// TIA Portal V17 export
// export: Created 2025-08-05T09:36:00.9032134Z, ExportSetting WithDefaults, DisplayName Totally Integrated Automation Portal, DisplayVersion V17, DisplayName TIA Portal Openness, DisplayVersion V17, DisplayName TIA Portal Version Control Interface, DisplayVersion V17, DisplayName SINAMICS Startdrive Advanced, DisplayVersion V17, DisplayName SINAMICS Startdrive G130, G150, S120, S150, SINAMICS MV, S210, DisplayVersion V17, DisplayName SINAMICS Startdrive G110M, G120, G120C, G120D, G120P, G115D, DisplayVersion V17, DisplayName STEP 7 Professional, DisplayVersion V17, DisplayName STEP 7 Safety, DisplayVersion V17, DisplayName WinCC Advanced, DisplayVersion V17
TYPE "typeTeststoppSBTPopUpWarn"
// V 01.00
// stored: IsFailsafeCompliant false
   STRUCT
      DoNotOpenSafeGuard : Bool;   // Bremsentest/Teststopp aktiv => Schutzeinrichtung nicht unterbrechen/öffnen / Brake test/test stop active => do not interrupt/open safeguard
      SafeGuardNotOpen { S7_SetPoint := 'True'} : Bool := false;   // Bremsentest/Teststopp angefordert => Schutzeinrichtung kann nicht geöffnet/entriegelt werden (Leistung ein oder E2 erforderlich) / Brake test/test stop requested => safeguard cannot be opened/unlocked (power on or E2 required)
      BrakeTestImmediately { S7_SetPoint := 'True'} : Bool := false;   // Schutzeinrichtung für Bremsentest/Teststopp schließen oder quittieren / Close or acknowledge safeguard for brake test/test stop
      BrakeTestNioPowerOff { S7_SetPoint := 'True'} : Bool := false;   // Bremsentest nio => Leistung aus (Bremse/Antrieb austauschen) / Brake test NOK => power off (exchange brake/drive)
      BrakeTestOnlyInHome : Bool;   // Bremsentest/Teststopp ist nur in Grundstellung möglich / Brake test/test stop only possible in home position
   END_STRUCT;
END_TYPE
